// TIA Portal V16 export
// export: Created 2024-09-05T17:36:34.5845061Z, ExportSetting WithDefaults, DisplayName Totally Integrated Automation Portal, DisplayVersion V16 Update 6, DisplayName TIA Portal Version Control Interface, DisplayVersion V16 Update 2, DisplayName TIA Portal Openness, DisplayVersion V16 Update 6, DisplayName STEP 7 Professional, DisplayVersion V16 Update 6, DisplayName STEP 7 Safety, DisplayVersion V16, DisplayName WinCC Advanced, DisplayVersion V16 Update 6
VAR_GLOBAL   // PLC tag table "DM_SM_RH"
   "DM_SMRH-TriggerEnable" AT %Q13.0 : Bool;
   "DM_SMRH-Trigger" AT %Q13.1 : Bool;
   "DM_SMRH-TriggerReady" AT %I29.0 : Bool;
   "DM_SMRH-TriggerAck" AT %I29.1 : Bool;
   "DM_SMRH-Acquiring" AT %I29.2 : Bool;
   "DM_SMRH-MissedAcq" AT %I29.3 : Bool;
   "DM_SMRH-TriggerID" AT %IW30 : Word;
   "DM_SMRH-BufferResultsEnable" AT %Q14.0 : Bool;
   "DM_SMRH-ResultsAck" AT %Q14.1 : Bool;
   "DM_SMRH-Decoding" AT %I18.0 : Bool;
   "DM_SMRH-Decode Complete" AT %I18.1 : Bool;
   "DM_SMRH-Results Buffer Overrun" AT %I18.2 : Bool;
   "DM_SMRH-Results Available" AT %I18.3 : Bool;
   "DM_SMRH-General Fault" AT %I18.7 : Bool;
   "DM_SMRH-Train Code" AT %Q15.0 : Bool;
   "DM_SMRH-Train Match String" AT %Q15.1 : Bool;
   "DM_SMRH-Train Focus" AT %Q15.2 : Bool;
   "DM_SMRH-Train Brightness" AT %Q15.3 : Bool;
   "DM_SMRH-Untrain" AT %Q15.4 : Bool;
   "DM_SMRH-Execute DMCC" AT %Q15.6 : Bool;
   "DM_SMRH-Set Match String" AT %Q15.7 : Bool;
   "DM_SMRH-Train Code Ack" AT %I19.0 : Bool;
   "DM_SMRH-Train Match String Ack" AT %I19.1 : Bool;
   "DM_SMRH-Train Focus Ack" AT %I19.2 : Bool;
   "DM_SMRH-Train Brightness Ack" AT %I19.3 : Bool;
   "DM_SMRH-Untrain Ack" AT %I19.4 : Bool;
   "DM_SMRH-Execute DMCC Ack" AT %I19.6 : Bool;
   "DM_SMRH-Set Match String Ack" AT %I19.7 : Bool;
   "DM_SMRH-UserData Option" AT %QW332 : Word;
   "DM_SMRH-UserData Length" AT %QW334 : Word;
   "DM_SMRH-UserData[0]" AT %QB336 : Byte;
   "DM_SMRH-UserData[1]" AT %QB337 : Byte;
   "DM_SMRH-UserData[2]" AT %QB338 : Byte;
   "DM_SMRH-UserData[3]" AT %QB339 : Byte;
   "DM_SMRH-UserData[4]" AT %QB340 : Byte;
   "DM_SMRH-UserData[5]" AT %QB341 : Byte;
   "DM_SMRH-UserData[6]" AT %QB342 : Byte;
   "DM_SMRH-UserData[7]" AT %QB343 : Byte;
   "DM_SMRH-UserData[8]" AT %QB344 : Byte;
   "DM_SMRH-UserData[9]" AT %QB345 : Byte;
   "DM_SMRH-UserData[10]" AT %QB346 : Byte;
   "DM_SMRH-UserData[11]" AT %QB347 : Byte;
   "DM_SMRH-UserData[12]" AT %QB348 : Byte;
   "DM_SMRH-UserData[13]" AT %QB349 : Byte;
   "DM_SMRH-UserData[14]" AT %QB350 : Byte;
   "DM_SMRH-UserData[15]" AT %QB351 : Byte;
   "DM_SMRH-ResultID" AT %IW528 : Word;
   "DM_SMRH-Result Code" AT %IW530 : Word;
   "DM_SMRH-Result Extended" AT %IW532 : Word;
   "DM_SMRH-Result Length" AT %IW534 : Word;
   "DM_SMRH-InspectionResults[0]" AT %IB536 : Byte;
   "DM_SMRH-InspectionResults[1]" AT %IB537 : Byte;
   "DM_SMRH-InspectionResults[2]" AT %IB538 : Byte;
   "DM_SMRH-InspectionResults[3]" AT %IB539 : Byte;
   "DM_SMRH-InspectionResults[4]" AT %IB540 : Byte;
   "DM_SMRH-InspectionResults[5]" AT %IB541 : Byte;
   "DM_SMRH-InspectionResults[6]" AT %IB542 : Byte;
   "DM_SMRH-InspectionResults[7]" AT %IB543 : Byte;
   "DM_SMRH-InspectionResults[8]" AT %IB544 : Byte;
   "DM_SMRH-InspectionResults[9]" AT %IB545 : Byte;
   "DM_SMRH-InspectionResults[10]" AT %IB546 : Byte;
   "DM_SMRH-InspectionResults[11]" AT %IB547 : Byte;
   "DM_SMRH-InspectionResults[12]" AT %IB548 : Byte;
   "DM_SMRH-InspectionResults[13]" AT %IB549 : Byte;
   "DM_SMRH-InspectionResults[14]" AT %IB550 : Byte;
   "DM_SMRH-InspectionResults[15]" AT %IB551 : Byte;
END_VAR
